{attribute 'GeneratedUsingTerminal: KL1002'}
{attribute addProperty BoxType "KL1002"}
{attribute addProperty Id "InputAT %I*BOOL0"}
{attribute addProperty CRC "2278121078"}
{attribute addProperty Size "0"}
TYPE Channel_87C95E76 EXTENDS InputBase_8311D824 :
STRUCT
	{attribute addProperty Name "Input"}
	Input AT %I* : BOOL;
END_STRUCT
END_TYPE

(* stored: Version 1.2.0.0, ProductVersion 3.1.4024.9
   DUT Channel_87C95E76: Id {6b93171d-44fc-40d9-aab6-14d98b2dcf45} *)
